// TIA Portal V18 export
// export: Created 2026-03-12T15:56:20.3291369Z, ExportSetting WithDefaults, DisplayName Totally Integrated Automation Portal, DisplayVersion V18 Update 5, DisplayName TIA Portal Openness, DisplayVersion V18 Update 5, DisplayName TIA Portal Version Control Interface, DisplayVersion V18, DisplayName SINAMICS Startdrive Advanced, DisplayVersion V18, DisplayName SINAMICS Startdrive G130, G150, S120, S150, SINAMICS MV, S210, DisplayVersion V18, DisplayName SINAMICS Startdrive G110M, G120, G120C, G120D, G120P, G115D, DisplayVersion V18, DisplayName STEP 7 Professional, DisplayVersion V18 Update 5, DisplayName STEP 7 Safety, DisplayVersion V18, DisplayName WinCC Professional, DisplayVersion V18 Update 5
DATA_BLOCK "FB MODOS DE OPERAÇÃO BH-01B"   // DB218
VERSION : 0.1
// stored: AutoNumber true, DBAccessibleFromOPCUA true, DBAccessibleFromWebserver true, InstanceOfName FB MODOS DE OPERAÇÃO, InstanceOfType FB
"FB MODOS DE OPERAÇÃO"
   // VAR_INPUT
   //    INPUT_RM : Bool;
   //    INPUT_RA : Bool;
   //    INPUT_LM : Bool;
   //    INPUT_LA : Bool;
   // END_VAR
   // VAR_OUTPUT
   //    OUTPUT_MODO : Int;
   // END_VAR
BEGIN
END_DATA_BLOCK
